VAR_GLOBAL CONSTANT
	udiMax_CylinderNum : UDINT := 53;
END_VAR

(* stored: Version 1.1.0.1, ProductVersion 3.1.4024.13
   GVL GVL_Machine_Const: Id {9386644b-2565-4100-ba97-6589634c725e} *)
